// Calvin - E_OffOn
// Rev 1.00 - March 23, 2023

TYPE E_OffOn :
(
	eOFF 	:= 1,
	eON		:= 2
);
END_TYPE

(* stored: Version 1.1.0.1, ProductVersion 3.1.4024.12
   DUT E_OffOn: Id {b133d4d2-053f-4b92-913e-ed12b077ddd7} *)
